FUNCTION_BLOCK CompositeBlockWithoutConnections
  FBS
    BaseBlock1 : BaseBlock;
    EA_2_router : EA_2_router;
    EA_network1_0 : EA_network1;
    EA_network1_1 : EA_network1;
    EA_LeftPublishSubscribeAdapter_0 : EA_LeftPublishSubscribeAdapter;
    Publish_Left_EA_0 : PUBLISH_5;
    Subscribe_Left_EA_0 : SUBSCRIBE_5;
    EA_LeftPublishSubscribeAdapter_1 : EA_LeftPublishSubscribeAdapter;
    Publish_Left_EA_1 : PUBLISH_5;
    Subscribe_Left_EA_1 : SUBSCRIBE_5;
  END_FBS
  EVENT_CONNECTIONS
    EA_LeftPublishSubscribeAdapter_0.REQ TO Publish_Left_EA_0.REQ;
    Subscribe_Left_EA_0.IND TO EA_LeftPublishSubscribeAdapter_0.IND;
    EA_LeftPublishSubscribeAdapter_1.REQ TO Publish_Left_EA_1.REQ;
    Subscribe_Left_EA_1.IND TO EA_LeftPublishSubscribeAdapter_1.IND;
  END_CONNECTIONS
  DATA_CONNECTIONS
    EA_LeftPublishSubscribeAdapter_0.I_E_number TO Publish_Left_EA_0.SD_1;
    EA_LeftPublishSubscribeAdapter_0.O_data1 TO Publish_Left_EA_0.SD_2;
    EA_LeftPublishSubscribeAdapter_0.O_data2 TO Publish_Left_EA_0.SD_3;
    EA_LeftPublishSubscribeAdapter_0.N_I_data1 TO Publish_Left_EA_0.SD_4;
    EA_LeftPublishSubscribeAdapter_0.N_I_data2 TO Publish_Left_EA_0.SD_5;
    Subscribe_Left_EA_0.RD_1 TO EA_LeftPublishSubscribeAdapter_0.O_E_number;
    Subscribe_Left_EA_0.RD_2 TO EA_LeftPublishSubscribeAdapter_0.I_data1;
    Subscribe_Left_EA_0.RD_3 TO EA_LeftPublishSubscribeAdapter_0.I_data2;
    Subscribe_Left_EA_0.RD_4 TO EA_LeftPublishSubscribeAdapter_0.N_O_data1;
    Subscribe_Left_EA_0.RD_5 TO EA_LeftPublishSubscribeAdapter_0.N_O_data2;
    EA_LeftPublishSubscribeAdapter_1.I_E_number TO Publish_Left_EA_1.SD_1;
    EA_LeftPublishSubscribeAdapter_1.O_data1 TO Publish_Left_EA_1.SD_2;
    EA_LeftPublishSubscribeAdapter_1.O_data2 TO Publish_Left_EA_1.SD_3;
    EA_LeftPublishSubscribeAdapter_1.N_I_data1 TO Publish_Left_EA_1.SD_4;
    EA_LeftPublishSubscribeAdapter_1.N_I_data2 TO Publish_Left_EA_1.SD_5;
    Subscribe_Left_EA_1.RD_1 TO EA_LeftPublishSubscribeAdapter_1.O_E_number;
    Subscribe_Left_EA_1.RD_2 TO EA_LeftPublishSubscribeAdapter_1.I_data1;
    Subscribe_Left_EA_1.RD_3 TO EA_LeftPublishSubscribeAdapter_1.I_data2;
    Subscribe_Left_EA_1.RD_4 TO EA_LeftPublishSubscribeAdapter_1.N_O_data1;
    Subscribe_Left_EA_1.RD_5 TO EA_LeftPublishSubscribeAdapter_1.N_O_data2;
  END_CONNECTIONS
  ADAPTER_CONNECTIONS
    BaseBlock1.plug TO EA_2_router.socket;
    EA_2_router.plug_0 TO EA_network1_0.Socket_Connection;
    EA_2_router.plug_1 TO EA_network1_1.Socket_Connection;
    EA_network1_0.Plug_Connection TO EA_LeftPublishSubscribeAdapter_0.socket;
    EA_network1_1.Plug_Connection TO EA_LeftPublishSubscribeAdapter_1.socket;
  END_CONNECTIONS
END_FUNCTION_BLOCK
